# EPICS substitutions: EUROTHRM/EUROTHRM-IOC-01App/Db/unit_setter.substitutions
file $(UTILITIES)/db/unit_setter.template {
  pattern
    {P,    FROM, TO, PROCESS_FLAGS}

    {"\$(P)", "UNITS", "TEMP", "PP"}
    {"\$(P)", "UNITS", "TEMP:SP", ""}
    {"\$(P)", "UNITS", "TEMP:SP:RBV", "PP"}
}
